{attribute 'qualified_only'}
{attribute 'strict'}
TYPE State_Vereinzelung :
(
	Off,
	Check,
	Init,
	Init_wait,
	Bereit,	
	Auswerfen,
	Auswerfen_wait,
	Fertig
);
END_TYPE

(* stored: Version 1.1.0.1, ProductVersion 3.1.4024.12
   DUT State_Vereinzelung: Id {30bc5d47-45ca-449f-8883-a2289c180bb0} *)
